FUNCTION_BLOCK LinearEncodedDrive_3Sensor EXTENDS FBA_LinearDrive IMPLEMENTS I_LinearEncodedDrive
VAR_INPUT
	drive : I_EncodedDrive;
	homeAt0 : BOOL;
	allowDualSideTraverse : BOOL; //allows motion between home to retractLimit
END_VAR
VAR_OUTPUT
	position : LREAL;
	velocity : LREAL;
END_VAR
VAR
	extendLimit AT %I* : BOOL;
	retractLimit AT %I* : BOOL;
	
	homePosition : LREAL;
	limitPosition : LREAL;
	
	calculation : (IDLE, EXTEND, RETRACT, CALCULATE, DONE);
END_VAR

override();

ready := bEnable AND NOT Active AND HomeSet;

PROPERTY Active : BOOL
GET
Active := drive.Active;
END_GET
END_PROPERTY

PROPERTY AtExtendLimit : BOOL
GET
AtExtendLimit := extendLimit <> sensorDefaultState;
END_GET
END_PROPERTY

PROPERTY AtRetractLimit : BOOL
GET
AtRetractLimit := retractLimit <> sensorDefaultState;
END_GET
END_PROPERTY

METHOD PRIVATE calculatePositions : BOOL
(*
THIS METHOD IS ONLY TO BE CALLED IF homeAt0 IS FALSE

not all drives have their home sensor at the 0 position
the purpose of this method is to calculate the home position, under the assumption that the extend limit sensor is 0

implementation:
	start from home
	reach the extend limit and set position to 0
	return to the home sensor and set the home position to the current position
*)
CASE calculation OF
	IDLE:
		calculation := EXTEND;
		
	EXTEND:		
		IF AtExtendLimit THEN
			
			IF homeAt0 THEN
				limitPosition := CurrentPosition;
				calculation := RETRACT;
			
			ELSIF setPosition(newPosition := 0) THEN
				limitPosition := 0;
				calculation := RETRACT;
			END_IF
		
		ELSE
			moveContinuous(newDirection := MC_Negative_Direction);
		END_IF
		
	RETRACT:
		IF AtHome THEN
			
			IF homeAt0 THEN
				homePosition := 0;
				calculation := DONE;
			
			ELSE
				homePosition := CurrentPosition;
				calculation := DONE;
			END_IF
		
		ELSE
			moveContinuous(newDirection := MC_Positive_Direction);
		END_IF
		
	DONE:
		calculation := 0;
		calculatePositions := TRUE;
		
END_CASE
END_METHOD

PROPERTY CurrentPosition : LREAL
GET
CurrentPosition := position;
END_GET
END_PROPERTY

PROPERTY Error : BOOL
GET
error := drive.Error;
END_GET
END_PROPERTY

METHOD homingSequence : BOOL
(*
homing sequence is different for linear motion devices with limit sensors
*)
CASE step OF
	Homing.IDLE:
		reset();
		IF bEnable THEN
			step := Homing.RETRY;
		END_IF
		
	Homing.START:
		IF AtHome THEN
			step := Homing.STOP;
			
		ELSIF AtRetractLimit THEN
			step := Homing.RETRY;
			
		ELSE
			moveContinuous(newDirection:= MC_Positive_Direction);
		END_IF
		
	Homing.RETRY:
		IF AtExtendLimit THEN
			step := Homing.START;
		ELSE
			moveContinuous(newDirection:= MC_Positive_Direction);
		END_IF
		
	Homing.STOP:
		IF stop() THEN
			step := Homing.SET;
		END_IF
		
	Homing.SET:
		IF calculatePositions() THEN
			step := Homing.DONE;
		END_IF
		
	Homing.DONE:
		homingComplete := TRUE;
		step := Homing.IDLE;
		
END_CASE
END_METHOD

METHOD moveAbsolute : BOOL
VAR_INPUT
	newTarget : LREAL;
END_VAR
(*
VAR_OUTPUT
	fault : BOOL;
END_VAR
*)
drive.moveAbsolute(newTarget:= newTarget);

moveAbsolute := drive.CurrentPosition = newTarget;
END_METHOD

METHOD moveContinuous : BOOL
VAR_INPUT
	//direction : BOOL; //direction (F = inwards, T = outwards)
	newDirection : MC_Direction;
END_VAR
drive.moveContinuous(newDirection:= newDirection);

direction := newDirection;
END_METHOD

METHOD moveRelative : BOOL
VAR_INPUT
	distance : LREAL;
END_VAR
drive.moveRelative(distance:= distance);
END_METHOD

METHOD PRIVATE override : BOOL
VAR_INPUT
END_VAR
(*
-at home and attempting to traverse outward
-at outer limit and attempting to traverse outward
-at inner limit and attempting to traverse inwards
*)
(*
inward = negative direction, negative velocity
outward = positive direction, positive velocity
*)

IF error THEN
	stop();
	reset();
	
ELSIF
	(NOT allowDualSideTraverse AND AtHome AND (TargetPosition > CurrentPosition OR direction = MC_Positive_Direction)) OR
	(AtExtendLimit AND (TargetPosition > CurrentPosition OR direction = MC_Negative_Direction)) OR
	(AtRetractLimit AND (TargetPosition < CurrentPosition OR direction = MC_Positive_Direction))
THEN
	stop();
END_IF
END_METHOD

METHOD reset : BOOL
VAR_INPUT
END_VAR
reset := drive.reset();
END_METHOD

METHOD setPosition : BOOL
VAR_INPUT
	newPosition : LREAL;
END_VAR
setPosition := drive.setPosition(newPosition:= newPosition);
END_METHOD

METHOD stop : BOOL
VAR_INPUT
END_VAR
drive.stop();
END_METHOD

PROPERTY TargetPosition : LREAL
GET
END_GET
END_PROPERTY

METHOD toHome : BOOL
VAR_INPUT
END_VAR
moveAbsolute(newTarget := homePosition);
END_METHOD

END_FUNCTION_BLOCK

(* stored: Version 1.1.0.1, ProductVersion 3.1.4024.11
   POU LinearEncodedDrive_3Sensor: Id {761e1ca8-c594-4778-a3ee-320c485e47c5}, SpecialFunc None
   Folder Private: Id {bd86a63a-379c-495a-b631-1ebf263b2583}
   Folder Properties: Id {0665c6da-7d70-40c1-ba4f-a5532fff129a}
   Property Active: Id {481eda0f-e6fa-4837-8913-47f58ff9e1d1}
   Get Get: Id {83394e4f-e6eb-47b9-81b2-58fce67b6ddb}
   Property AtExtendLimit: Id {e730bcc5-cd9f-4bd1-a73b-47808ca5218d}
   Get Get: Id {6862abe5-0ff8-494d-afdd-b365d8adac81}
   Property AtRetractLimit: Id {5c5a9b2a-dfa2-490d-a9d7-ee69d2a6fa32}
   Get Get: Id {1b01b7c1-f2d0-468c-bb80-102d8acef053}
   Method calculatePositions: Id {0f65d4ca-e52f-47a4-9127-3fad98c26602}
   Property CurrentPosition: Id {42368fde-8acb-4716-8c79-a0e8c7a1c3e2}
   Get Get: Id {26490d82-7c62-4aa3-810b-81bdc6f93127}
   Property Error: Id {7e78b592-6e07-43e9-b48c-1dd6da2a5a8c}
   Get Get: Id {7b328bcb-8cb3-4a4b-954b-76ad51e7e1e0}
   Method homingSequence: Id {6dbeac1c-ebf9-4cc2-ad7d-db1135768e34}
   Method moveAbsolute: Id {3f9c4462-6669-486c-85e2-4d66abb58623}
   Method moveContinuous: Id {0e9a34c9-962d-4fbb-8ed2-7b42fd682577}
   Method moveRelative: Id {04ca0e88-1400-4101-a6c1-df72f68aaf4c}
   Method override: Id {bddd7bd6-f146-447d-a29a-c7ee59c0d2ad}
   Method reset: Id {f29d8bf4-36b5-48f3-8aba-1d0cad9fe926}
   Method setPosition: Id {506bee99-6621-4aa4-be49-cabca1cca014}
   Method stop: Id {33abe24c-d7fd-4671-8b51-407b6cd4373f}
   Property TargetPosition: Id {97f34255-16f9-414c-95cc-2a8a1f1f29e0}
   Get Get: Id {852785ec-3dca-4489-bbe6-beac91a0c354}
   Method toHome: Id {d98fdb48-bfe6-4ed5-971f-39643682a9f3} *)
